// TIA Portal V18 export
TYPE "LGasp_taglioValvProp"
// stored: IsFailsafeCompliant false
   STRUCT
      nomeprogramma : WString[30];   // nome del programma trasferito dal PC
      ID : DInt;   // ID del programma
      num_pressa : Int;   // numero della pressa selezionata
      num_pressa_old : Int;   // appoggio numero della pressa selezionata
      scrittura_prg : Bool;   // 1=programma/modifiche trasferite
      pms : Struct   // dati del punto morto superiore in mm del programma automatico [mm]
         limitemin : LReal;   // da PLC
         limitemax : LReal := 1000.0;   // da PLC
         valore : LReal;   // da programma PC
      END_STRUCT;
      pmi : Struct   // dati del punto morto inferiore in mm del programma automatico [mm]
         limitemin : LReal;   // da PLC
         limitemax : LReal := 1000.0;   // da PLC
         valore : LReal;   // da programma PC
      END_STRUCT;
      pos_cambiostampo : Struct   // dati per posizione cambio stampo [mm]
         enablevis : Bool;   // da PLC, abilita il campo nella pagina del PC
         limitemin : LReal;   // da PLC
         limitemax : LReal := 1000.0;   // da PLC
         valore : LReal;   // da programma PC
      END_STRUCT;
      speed_discesa : Struct   // dati della velocità di discesa [%] del programma automatico
         limitemin : LReal;   // da PLC
         limitemax : LReal := 1000.0;   // da PLC
         valore : LReal;   // da programma PC / %
      END_STRUCT;
      speed_salita : Struct   // dati della velocità di salita [%] del programma automatico
         limitemin : LReal;   // da PLC
         limitemax : LReal := 1000.0;   // da PLC
         valore : LReal;   // da programma PC / %
      END_STRUCT;
      speed_manuale : Struct   // dati della velocità in manuale [%]
         limitemin : LReal;   // da PLC
         limitemax : LReal := 1000.0;   // da PLC
         valore : LReal;   // da programma PC / %
      END_STRUCT;
      accelerazione : Struct   // dati accelerazione [mm/sec2]
         enablevis : Bool;   // da PLC, abilita il campo nella pagina del PC
         limitemin : LReal;   // da PLC
         limitemax : LReal := 1000.0;   // da PLC
         valore : LReal;   // da programma PC / mm/sec2
      END_STRUCT;
      decelerazione : Struct   // dati decelerazione [mm/sec2]
         enablevis : Bool;   // da PLC, abilita il campo nella pagina del PC
         limitemin : LReal;   // da PLC
         limitemax : LReal := 1000.0;   // da PLC
         valore : LReal;   // da programma PC / mm/sec2
      END_STRUCT;
      area_peh : Struct   // finestra di tolleranza posizione valvola in quota [mm]
         limitemin : LReal;   // da PLC
         limitemax : LReal := 1000.0;   // da PLC
         valore : LReal;   // da programma PC / mm
      END_STRUCT;
      inerzia_pos : Struct   // inerzia positiva [mm]
         limitemin : LReal;   // da PLC
         limitemax : LReal := 1000.0;   // da PLC
         valore : LReal;   // da programma PC / mm
      END_STRUCT;
      inerzia_neg : Struct   // inerzia negativa [mm]
         limitemin : LReal;   // da PLC
         limitemax : LReal := 1000.0;   // da PLC
         valore : LReal;   // da programma PC / mm
      END_STRUCT;
      forza : Struct   // in % del valore massimo
         enable : Bool;   // abilita controllo di forza da PC
         limitemin : LReal;   // da PLC
         limitemax : LReal := 1000.0;   // da PLC
         valore : LReal;   // da programma PC in % / %
      END_STRUCT;
      vis : Struct   // dati di visualizzazione
         nome : WString[30];   // nome fisso nel PLC e visualizzato dal PC
         temposalita : LReal;   // sec.
         tempodiscesa : LReal;   // sec.
         tempototale : LReal;   // sec.
         posattuale : LReal;   // mm
         pms_max : LReal;   // Quota massima del PMS mm (dipende dalla meccanica, dato fisso nel PLC) / mm
         pmi_max : LReal;   // Quota massima del PMI mm (dipende dalla meccanica, dato fisso nel PLC) / mm
         pmi_ciclo : LReal;   // Valore PMI raggiunto durante il ciclo, utile per calcolare inerzia / mm
         speed_max : LReal;   // Velocità massima [mm/s] scritta da plc / mm/sec
         speedattuale : LReal;   // mm/sec
         forza_max : LReal;   // KN / kilo-newton
         forzaattuale : LReal;   // kilo-newton / KN
         controlloForzaON : Bool;   // controllo di forza limite raggiunto / controllo di forza in funzione
         peh : Bool;   // in tolleranza
         pms : Bool;   // in pos pms max
         pmi : Bool;   // in pos pmi max
         flt : Bool;   // in errore
      END_STRUCT;
   END_STRUCT;
END_TYPE
